Fanuc KAREL source: ka00227.KL

-- PROVISIONAL review KL for V1013-1; original PC SHA256 d69e33b3ba882a4e052b6c95df782032ae63c05a374939e87d3a7b2d7a1a96b3
-- Incomplete behavior may be omitted. Consult companion uncertainty JSON. Do not deploy.
PROGRAM KA00227
%NOLOCKGROUP
-- UNRESOLVED_DECL SRC type=001100
-- UNRESOLVED_DECL DST type=001100
BEGIN
  -- UNRESOLVED_PC offsets 5-20; opcodes 22,22,30
  -- UNRESOLVED_PC offsets 25-29; opcodes 7F
END KA00227
